PROGRAM MAIN
VAR
END_VAR

END_PROGRAM

(* stored: Version 1.1.0.1
   POU MAIN: Id {e9c52344-6699-4725-9bd9-6c8454ddf2eb} *)
